{attribute 'GeneratedUsingTerminal: EK1122-0000-0018'}
{attribute addProperty BoxType "EK1122-0000-0018"}
{attribute addProperty Id "Beckhoff_EL1xxxsub_EK1100EK1100_AB5A94672"}
{attribute addProperty CRC "2737608987"}
{attribute addProperty Size "2"}
TYPE Beckhoff_EL1xxxEK1122_A32C991B EXTENDS EK1122_AB5A9467 :
STRUCT
	{attribute addProperty Name "Beckhoff_EL1xxxsub_EK1100"}
	{attribute addProperty PreviousPort "Beckhoff EL1xxxEK1122 : D"}
	Beckhoff_EL1xxxsub_EK1100 : EK1100_AB5A9467;
END_STRUCT
END_TYPE

(* stored: Version 1.2.0.0, ProductVersion 3.1.4024.9
   DUT Beckhoff_EL1xxxEK1122_A32C991B: Id {9b51aacd-d966-4510-a28f-3d4b2cd20eab} *)
